FUNCTION_BLOCK PAMFlowmeter EXTENDS PAProcessModule
VAR_INPUT
END_VAR
VAR_OUTPUT
END_VAR
VAR
	_PAPointMatIn1 : PAPoint(THIS^);
	_PAPointMatOut1 : PAPoint(THIS^);
END_VAR

METHOD FB_init : BOOL
VAR_INPUT
	bInitRetains : BOOL; // if TRUE, the retain variables are initialized (warm start / cold start)
	bInCopyCode : BOOL;  // if TRUE, the instance afterwards gets moved into the copy code (online change)
	parent : IACComponent;
END_VAR
AddPoint(_PAPointMatIn1);
AddPoint(_PAPointMatOut1);
END_METHOD

PROPERTY PUBLIC PAPointMatIn1 : IACPoint
GET
PAPointMatIn1 := _PAPointMatIn1;
END_GET
END_PROPERTY

PROPERTY PUBLIC PAPointMatOut1 : IACPoint
GET
PAPointMatOut1 := _PAPointMatOut1;
END_GET
END_PROPERTY

END_FUNCTION_BLOCK

(* stored: Version 1.1.0.1, ProductVersion 3.1.4020.12
   POU PAMFlowmeter: Id {aeb2f9a5-b5a7-43c3-a864-e642fd10288b}, SpecialFunc None
   Method FB_init: Id {17263f4f-dbb5-4ca8-88be-54ef5e190904}
   Property PAPointMatIn1: Id {426810ef-faf0-4473-a3e1-717c31bd15b1}
   Get Get: Id {d8803b1f-fdb3-4b58-86f7-a1696fa36bf2}
   Property PAPointMatOut1: Id {3bc6041d-96ae-4f05-803d-260b9f7a3524}
   Get Get: Id {e86a7ffd-bfc4-4845-a7c8-613c4d5cd6b4} *)
